FUNCTION_BLOCK MyFunctionBlock
VAR
END_VAR

END_FUNCTION_BLOCK

(* stored: Version 1.1.0.1, ProductVersion 3.1.4024.12
   POU MyFunctionBlock: Id {f883b766-d260-43ce-938d-9fd5a4142915}, SpecialFunc None *)
